FUNCTION_BLOCK MockDeserializableUserObject IMPLEMENTS I_Deserializable
VAR
	_name : STRING;
	_age : INT;
END_VAR

PROPERTY PUBLIC Age : INT
GET
Age := _age;
END_GET
SET
_age := Age;
END_SET
END_PROPERTY

PROPERTY PUBLIC Name : STRING
GET
Name := _name;
END_GET
SET
_name := Name;
END_SET
END_PROPERTY

METHOD TryDeserializeFrom : BOOL
VAR_INPUT
	Deserializer : I_Deserializer;
END_VAR
TryDeserializeFrom := 
	Deserializer.TryGetKeyString('Name',_name) AND
	Deserializer.TryGetKeyInt('Age',_age);
END_METHOD

END_FUNCTION_BLOCK

(* stored: Version 1.1.0.1, ProductVersion 3.1.4024.12
   POU MockDeserializableUserObject: Id {ecd607bb-83a9-4d79-a8ab-363938f57e03}, SpecialFunc None
   Property Age: Id {bfc899d7-b9b5-43a3-b21c-921d9cb41d78}
   Get Get: Id {8b729a3d-1d76-409c-8a9f-bdac2d562b4f}
   Set Set: Id {b445f0fa-29e2-473e-95a1-e92418b1fd6e}
   Property Name: Id {8c5e2a62-b93f-4d2f-bf42-ec984f3a59c9}
   Get Get: Id {6f1599e5-a554-42cd-8e65-078b3108d65d}
   Set Set: Id {77a98b9d-145d-460f-9c55-6c4834ef40c6}
   Method TryDeserializeFrom: Id {1c9b47aa-03bf-4aca-bfd2-63a3b957b556} *)
